// Checks if value can be converted to string
FUNCTION F_ISANYSTRCOMPAT : BOOL
VAR_INPUT
	Value : ANY;
END_VAR

CASE Value.TypeClass OF
	__SYSTEM.TYPE_CLASS.TYPE_STRING,
	__SYSTEM.TYPE_CLASS.TYPE_WSTRING,
	__SYSTEM.TYPE_CLASS.TYPE_BOOL,
	__SYSTEM.TYPE_CLASS.TYPE_BYTE,
	__SYSTEM.TYPE_CLASS.TYPE_WORD,
	__SYSTEM.TYPE_CLASS.TYPE_DWORD,
	__SYSTEM.TYPE_CLASS.TYPE_LWORD,
	__SYSTEM.TYPE_CLASS.TYPE_SINT,
	__SYSTEM.TYPE_CLASS.TYPE_INT,
	__SYSTEM.TYPE_CLASS.TYPE_DINT,
	__SYSTEM.TYPE_CLASS.TYPE_LINT,
	__SYSTEM.TYPE_CLASS.TYPE_USINT,
	__SYSTEM.TYPE_CLASS.TYPE_UINT,
	__SYSTEM.TYPE_CLASS.TYPE_UDINT,
	__SYSTEM.TYPE_CLASS.TYPE_ULINT,
	__SYSTEM.TYPE_CLASS.TYPE_REAL,
	__SYSTEM.TYPE_CLASS.TYPE_LREAL,
	__SYSTEM.TYPE_CLASS.TYPE_TIME,
	__SYSTEM.TYPE_CLASS.TYPE_LTIME,
	__SYSTEM.TYPE_CLASS.TYPE_DATE,
	__SYSTEM.TYPE_CLASS.TYPE_DATEANDTIME,
	__SYSTEM.TYPE_CLASS.TYPE_TIMEOFDAY,
	__SYSTEM.TYPE_CLASS.TYPE_POINTER:
		F_ISANYSTRCOMPAT := TRUE;
ELSE
	RETURN;
END_CASE

END_FUNCTION

(* stored: Version 1.1.0.1, ProductVersion 3.1.4024.4
   POU F_ISANYSTRCOMPAT: Id {f8c9834e-b07b-40ff-91cc-a3ec005c552e}, SpecialFunc None *)
